FUNCTION_BLOCK FB_MC2_DigLockCtrl
VAR_INPUT
	bLockAxis			: BOOL;				(* set TRUE to lock axis, set FALSE to unlock axis *)
	fGearRatio			: LREAL;			(* gear ratio, can be changed on every PLC cycle *)
	sRamps				: ST_AxisCtrlRamps;	(* axis ramp structure *)
END_VAR
VAR_IN_OUT
	sAxisMaster			: AXIS_REF;			(* NC axis structure *)
	sAxisSlave			: AXIS_REF;			(* NC axis structure *)
END_VAR
VAR_OUTPUT
	bAxisLocked			: BOOL;				(* TRUE = cam locked *)
	bAxisError			: BOOL;				(* error occurred *)
	nAxisErrorID		: UDINT;			(* error code *)
	bAxisReady			: BOOL;
	bAxisUnlockPulse	: BOOL;				(* one-shot pulse output when slave is unlocked *)
END_VAR
VAR
	fbEnableLock		: RS;
	bEnableLock			: BOOL;
	fbGearIn			: MC_GearInDyn;
	fbGearOut			: MC_GearOut;
	bAxisInGear			: BOOL;
	bAxisActive			: BOOL;
	fbUnlockEvent		: F_TRIG;
	fbUnlockPulse		: TP;
END_VAR
(*
-------------------------------------------------------------------------------------------------
Date		Version	Author	Comments
-------------------------------------------------------------------------------------------------
30/01/2015	3.00.00	PB		No change

-------------------------------------------------------------------------------------------------
12/08/2013	1.11.00	PB		Bug fix - ControlLoopClosed for Slave also now cancels lock
05/02/2010	1.00.00	PB		Initial release

-------------------------------------------------------------------------------------------------
*)
VAR // added by the converter: edge detectors and wires of the graphical bodies
    _w1 : BOOL;
END_VAR

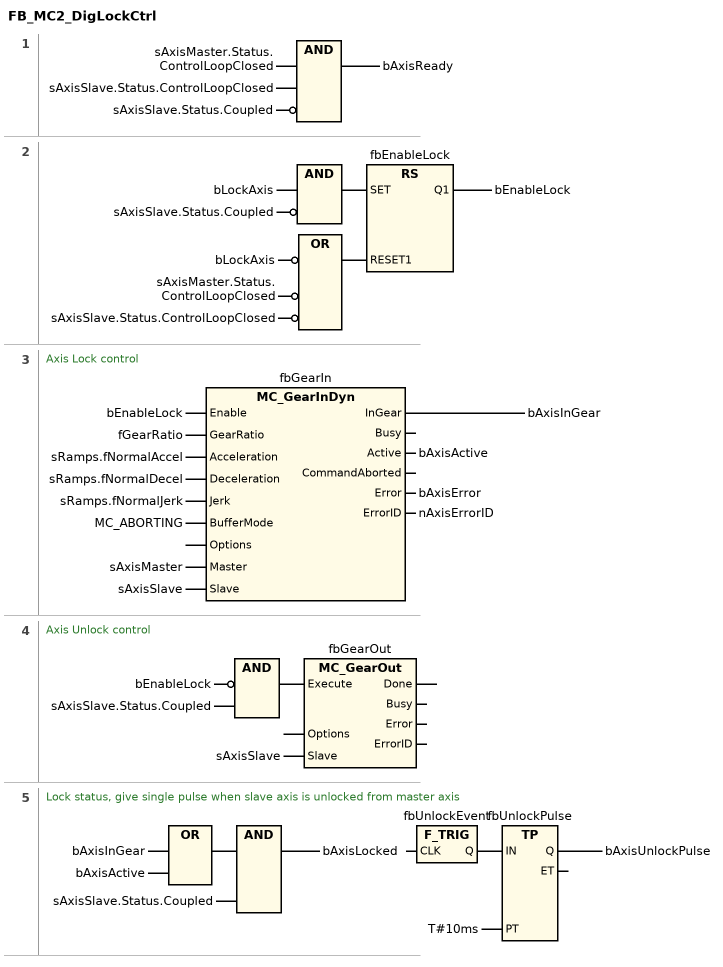
// NETWORK 1
bAxisReady := sAxisMaster.Status.ControlLoopClosed AND sAxisSlave.Status.ControlLoopClosed AND NOT sAxisSlave.Status.Coupled;

// NETWORK 2
fbEnableLock(SET := bLockAxis AND NOT sAxisSlave.Status.Coupled, RESET1 := NOT bLockAxis OR NOT sAxisMaster.Status.ControlLoopClosed OR NOT sAxisSlave.Status.ControlLoopClosed); // RS
bEnableLock := fbEnableLock.Q1;

// NETWORK 3
// Axis Lock control
fbGearIn(
    Enable := bEnableLock,
    GearRatio := fGearRatio,
    Acceleration := sRamps.fNormalAccel,
    Deceleration := sRamps.fNormalDecel,
    Jerk := sRamps.fNormalJerk,
    BufferMode := MC_ABORTING,
    Master := sAxisMaster,
    Slave := sAxisSlave,
    Active => bAxisActive,
    Error => bAxisError,
    ErrorID => nAxisErrorID); // MC_GearInDyn
bAxisInGear := fbGearIn.InGear;

// NETWORK 4
// Axis Unlock control
fbGearOut(Execute := NOT bEnableLock AND sAxisSlave.Status.Coupled, Slave := sAxisSlave); // MC_GearOut

// NETWORK 5
// Lock status, give single pulse when slave axis is unlocked from master axis
_w1 := (bAxisInGear OR bAxisActive) AND sAxisSlave.Status.Coupled;
bAxisLocked := _w1;
fbUnlockEvent(CLK := _w1); // F_TRIG
fbUnlockPulse(IN := fbUnlockEvent.Q, PT := T#10ms); // TP
bAxisUnlockPulse := fbUnlockPulse.Q;

END_FUNCTION_BLOCK

(* stored: Version 1.1.0.1, ProductVersion 3.1.4024.15
   POU FB_MC2_DigLockCtrl: Id {f4a659a3-8614-4fa2-af87-9a7122a8e94b}, SpecialFunc None *)
